FUNCTION_BLOCK MOD_StateIds (* OPC UA and local channel IDs of the module state manager *)
  (* Standard: 61499-2 *)
  (* Version 0.1, 2026-09-28, Project contributors, AAU Smart Production Lab *)
  PACKAGE modlib;
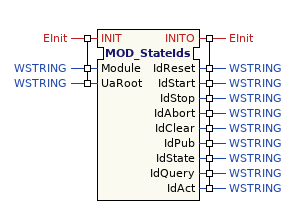
  EVENT_INPUT
    INIT : EInit WITH Module, UaRoot;
  END_EVENT
  EVENT_OUTPUT
    INITO : EInit WITH IdReset, IdStart, IdStop, IdAbort, IdClear, IdPub, IdState, IdQuery, IdAct;
  END_EVENT
  VAR_INPUT
    Module : WSTRING;
    UaRoot : WSTRING;
  END_VAR
  VAR_OUTPUT
    IdReset : WSTRING;
    IdStart : WSTRING;
    IdStop : WSTRING;
    IdAbort : WSTRING;
    IdClear : WSTRING;
    IdPub : WSTRING;
    IdState : WSTRING;
    IdQuery : WSTRING;
    IdAct : WSTRING;
  END_VAR
  EC_STATES
    INIT : INIT -> INITO;
  END_STATES
  ALGORITHM INIT IN ST:
IdReset := CONCAT(CONCAT(CONCAT("opc_ua[CREATE_METHOD;", CONCAT(UaRoot, "/Module/")), "Reset"), "]");
IdStart := CONCAT(CONCAT(CONCAT("opc_ua[CREATE_METHOD;", CONCAT(UaRoot, "/Module/")), "Start"), "]");
IdStop := CONCAT(CONCAT(CONCAT("opc_ua[CREATE_METHOD;", CONCAT(UaRoot, "/Module/")), "Stop"), "]");
IdAbort := CONCAT(CONCAT(CONCAT("opc_ua[CREATE_METHOD;", CONCAT(UaRoot, "/Module/")), "Abort"), "]");
IdClear := CONCAT(CONCAT(CONCAT("opc_ua[CREATE_METHOD;", CONCAT(UaRoot, "/Module/")), "Clear"), "]");
IdPub := CONCAT(CONCAT(CONCAT("opc_ua[WRITE;", CONCAT(UaRoot, "/Module/")), "State"), "]");
IdState := CONCAT(CONCAT("loc[", Module), "/state]");
IdQuery := CONCAT(CONCAT("loc[", Module), "/state/query]");
IdAct := CONCAT(CONCAT("loc[", Module), "/activity]");
  END_ALGORITHM
END_FUNCTION_BLOCK
